// TwinCAT 3 PLC project Green_Crane
// ProgramVersion: 3.1.4023.0
// libraries:
//   Tc2_Standard, * (Beckhoff Automation GmbH)
//   Tc2_System, * (Beckhoff Automation GmbH)
//   Tc3_Module, * (Beckhoff Automation GmbH)
// project tree:
//   DUTs/ E_Mode.TcDUT, ST_ActiveDamping.TcDUT
//   / GlobalTextList.TcGTLO, PlcTask.TcTTO, Visualization Manager.TcVMO (not stored)
//   GVLs/ G_Input.TcGVL, G_Output.TcGVL, G_Parameter.TcGVL
//   POUs/FBs/ FB_AutomaticControl.TcPOU, FB_Clock.TcPOU, FB_ManualControl.TcPOU, FB_SetMode.TcPOU
//   POUs/Imported FBs/ FB_CraneSimulator.TcPOU, FB_MotionReferenceGenerat.TcPOU, FB_ActiveDamping.TcPOU, FB_ClosedLoopControl.TcPOU, FB_OpenLoopControl.TcPOU, FB_ResetIntegralController.TcPOU
//   POUs/Programs/ MAIN.TcPOU (not stored), P_CraneControl.TcPOU
//   VISUs/ HMI.TcVIS
// real-time tasks:
//   TASK PlcTask: cycle T#10ms, priority 20, ADS port 350

CONFIGURATION Green_Crane
    RESOURCE PLC ON TwinCAT3
        TASK PlcTask(INTERVAL := T#10ms, PRIORITY := 20);
        PROGRAM MAIN WITH PlcTask : MAIN;
    END_RESOURCE
END_CONFIGURATION

// ---- DUTs/E_Mode.TcDUT
{attribute 'qualified_only'}
{attribute 'strict'}
TYPE E_Mode :
(
	Auto,
	Manual,
	Off
);
END_TYPE

// ---- DUTs/ST_ActiveDamping.TcDUT
TYPE ST_ActiveDamping :
STRUCT
	fFlowGainInverse : LREAL := 1.7153E03;	
	fHPF_Num1 : LREAL := 9.016E-12;
	fHPF_Num2 : LREAL := -9.016E-12;
	fHPF_Den1 : LREAL := 1.0;
	fHPF_Den2 : LREAL := -0.9905;
	fVDI_Num1 : LREAL := 25;
	fVDI_Num2 : LREAL := -48.83;
	fVDI_Num3 : LREAL := 23.85;
	fVDI_Den1 : LREAL := 1;
	fVDI_Den2 : LREAL := -1.721;
	fVDI_Den3 : LREAL := 0.7408;
END_STRUCT
END_TYPE

// ---- GVLs/G_Input.TcGVL
{attribute 'qualified_only'}
VAR_GLOBAL
	bPoweSwitch : BOOL;
	bOnOffSwitch : BOOL;
	bModeSwitch : BOOL;
	bStartSwitch : BOOL;
	bStopSwitch : BOOL;
	fJoyStickSignal : REAL;
END_VAR

// ---- GVLs/G_Output.TcGVL
{attribute 'qualified_only'}
VAR_GLOBAL
	sModeDisplay : STRING;
	bGreenLed : BOOL;
	bRedLed : BOOL;
	fOpenLoopControlOutput : LREAL;
	
END_VAR

// ---- GVLs/G_Parameter.TcGVL
{attribute 'qualified_only'}
VAR_GLOBAL
	fCycleTime : REAL := 0.01;
	fTime : REAL;
	eMode : E_Mode;
	fMaxVolumeFlow : REAL := 30.0;
	fCylinderSpeedRef : LREAL;
	
	
// MotionReference
	fStartPosition_m		: LREAL := 0.0;
	fStartVelocity_m		: LREAL	:= 0.0;
	fPositionSetpoint_ms	: LREAL := 0.25;
	fVelocitySetpoint_m		: LREAL := 0.025;
	fMaxPosition 			: LREAL := 0.45;
	fMinPosition 			: LREAL := 0.0;
	fMaxVelocity 			: LREAL := 0.05;
	fTimeBeforeStarting_s	: LREAL := 3.0;
	fRampTime_s				: LREAL := 1.0;
	fHoldPositionTime_s		: LREAL := 5.0;




// Automatic

	bEnableVelocityFeedForwardControl	: BOOL := TRUE;
	bEnableClosedLoopPositionControl	: BOOL := TRUE;
	bEnableIntegralController 			: BOOL := TRUE;
	bEnableActiveDamping 				: BOOL := TRUE;


// Closed Loop
	fMaxPositionError 					: LREAL := 1E-3;
	fProportionalGain 					: LREAL := 29.17;
	fIntegralGain 						: LREAL := 19.49;	
	
	
//Simulator

	bEnableSimulation					: BOOL := TRUE;
	
END_VAR

// ---- POUs/FBs/FB_AutomaticControl.TcPOU
FUNCTION_BLOCK FB_AutomaticControl
VAR_INPUT
	bEnable : BOOL;
	eMode : E_Mode;
	bStartSwitch : BOOL;
	bStopSwitch : BOOL;
END_VAR
VAR_OUTPUT
	fAutoOutput : LREAL;
END_VAR
VAR
	fbClock 						: FB_Clock;
	fbMotionReference 				: FB_MotionReferenceGenerat;
	fbVelocityFeedForwardControl 	: FB_OpenLoopControl;
	fbResetIntegralController		: FB_ResetIntegralController;
	fbClosedLoopControl		: FB_ClosedLoopControl;
	
	
	fStartPosition : LREAL;
	fStartVelocity : LREAL;
	fPositionSetpoint : LREAL;
	fVelocitySetpoint : LREAL;
	fTimeBeforeStarting : LREAL;
	fRampTime : LREAL;
	fHoldPositionTime : LREAL;

END_VAR

IF bEnable = FALSE THEN
	RETURN;
END_IF


fbClock(
	bStart := ((eMode = E_Mode.Auto) AND bStartSwitch = TRUE),
	bStop := bStopSwitch,
	fCycleTime := G_Parameter.fCycleTime,
);

fStartPosition := LIMIT(G_Parameter.fMinPosition, G_parameter.fStartPosition_m, G_Parameter.fMaxPosition);
fStartVelocity := LIMIT(0.0, G_parameter.fStartVelocity_m, G_parameter.fMaxVelocity );
fPositionSetpoint := LIMIT(G_Parameter.fMinPosition, G_Parameter.fPositionSetpoint_ms, G_Parameter.fMaxPosition);
fVelocitySetpoint := LIMIT(0.0, G_Parameter.fVelocitySetpoint_m, G_Parameter.fMaxVelocity);
fTimeBeforeStarting := LIMIT(0.0, G_Parameter.fTimeBeforeStarting_s, 10.0);
fRampTime := LIMIT(0.0, G_Parameter.fRampTime_s, 10.0);
fHoldPositionTime := LIMIT(0.0, G_Parameter.fHoldPositionTime_s, 60.0);

fbMotionReference(
	fStartposition_m := fStartPosition,
	fStartVelocity_m := fStartVelocity,
	fPositionSetpoint_ms := fPositionSetpoint,
	fVelocitySetpoint_m := fVelocitySetpoint,
	fTimeBeforeStarting_s := fTimeBeforeStarting,
	fRampTime_s := fRampTime,
	fHoldPositionTime_s := fHoldPositionTime,
	fClock_s := fbClock.fTimeInSeconds
);
	
	
fbVelocityFeedForwardControl(
	bEnable := G_Parameter.bEnableVelocityFeedForwardControl,
	fVelocityReference_ms := fbMotionReference.fVelocityReference_ms,
	fMaxValveFlow_lmin := G_Parameter.fMaxVolumeFlow
);
		
fbResetIntegralController(
	fVelocityReference_ms := fbMotionReference.fVelocityReference_ms,
	fPositionError_m := fbClosedLoopControl.fPositionError,
	fMaxPositionError_m := G_Parameter.fMaxPosition
);
	
	

fbClosedLoopControl(
	bEnable := G_Parameter.bEnableClosedLoopPositionControl,
	bActivateIntegralController := G_Parameter.bEnableIntegralController,
	bIntegralControllReset := fbResetIntegralController.bReset,
	fPositionFeedBack := 0.0,
	fProportionalGain := G_Parameter.fProportionalGain,
	fPositionReference := fbMotionReference.fPositionReference_m,
);
	
	IF (eMode = E_Mode.Auto AND G_input.bStartSwitch = TRUE) THEN
	fAutoOutput := LIMIT(-1.0, (fbVelocityFeedForwardControl.fVelocityFeedForward + fbClosedLoopControl.fClosedLoopPosition), 1.0);
ELSE
	fAutoOutput:= 0.0;
END_IF

END_FUNCTION_BLOCK

// ---- POUs/FBs/FB_Clock.TcPOU
FUNCTION_BLOCK FB_Clock
VAR_INPUT
	bStart : BOOL;
	bStop : BOOL;
	fCycleTime : REAL;
END_VAR
VAR_OUTPUT
	fTimeInSeconds : REAL;
END_VAR
VAR
END_VAR



IF bStart = TRUE AND bStop = FALSE THEN
	fTimeInSeconds := fTimeInSeconds + fCycleTime;
ELSE
	fTimeInSeconds := 0.0;
END_IF

END_FUNCTION_BLOCK

// ---- POUs/Imported FBs/FB_MotionReferenceGenerat.TcPOU
FUNCTION_BLOCK FB_MotionReferenceGenerat
VAR_INPUT
	fStartPosition_m: LREAL;
	fStartVelocity_m: LREAL;
	fPositionSetpoint_ms: LREAL;
	fVelocitySetpoint_m: LREAL;
	fTimeBeforeStarting_s: LREAL;
	fRampTime_s: LREAL;
	fHoldPositionTime_s: LREAL;
	fClock_s: LREAL;
END_VAR
VAR_OUTPUT
	fPositionReference_m: LREAL;
	fVelocityReference_ms: LREAL;
	fTotalMotionTime_s: LREAL;
	fErrorSignal: LREAL;
END_VAR
VAR
	Error: DINT;
	slopeExt: LREAL;
	slopeRetr: LREAL;
	tHold: LREAL;
	x1: LREAL;
	x4: LREAL;
	x1_tmp: LREAL;
	x1_tmp_tmp: LREAL;
	x4_tmp: LREAL;
	x4_tmp_tmp: LREAL;
	x4_tmp_tmp_0: LREAL;
	x1_tmp_0: LREAL;
END_VAR


(* Outputs for Atomic SubSystem: '<Root>/FB_MotionReferenceGenerator_nolimit' *)
(* MATLAB Function: '<S1>/WaveSignal' *)
(* MATLAB Function 'FB_MotionReferenceGenerator_nolimit/WaveSignal': '<S2>:1' *)
(* '<S2>:1:2' x_SP = x_ref - x0; *)
(* '<S2>:1:3' vs=v_ref; *)
(* '<S2>:1:4' slopeExt=v0-vs; *)
slopeExt := fStartVelocity_m - fVelocitySetpoint_m;
(* '<S2>:1:5' slopeRetr=-vs-v0; *)
slopeRetr := ( -fVelocitySetpoint_m) - fStartVelocity_m;
(* '<S2>:1:7' as = vs/tRamp; *)
(* '<S2>:1:8' s_acc=(vs^2-v0^2)/as; *)
(* '<S2>:1:10' tHold=(x_SP-s_acc)/vs; *)
tHold := ((fPositionSetpoint_ms - fStartPosition_m) - (((fVelocitySetpoint_m * fVelocitySetpoint_m) - (fStartVelocity_m * fStartVelocity_m)) / (fVelocitySetpoint_m / fRampTime_s))) / fVelocitySetpoint_m;
(* '<S2>:1:12' if tHold < 0 *)

IF tHold < 0.0 THEN 
    (* '<S2>:1:13' Error = 1; *)
    Error := 1;
ELSE 
    (* '<S2>:1:14' else *)
    (* '<S2>:1:15' Error = 0; *)
    Error := 0;
END_IF;

(* '<S2>:1:18' t1=tRamp; *)
(* '<S2>:1:19' t2=tHold; *)
(* '<S2>:1:20' t3=tRamp; *)
(* '<S2>:1:21' t4=tWait; *)
(* '<S2>:1:22' t5=t1; *)
(* '<S2>:1:23' t6=t2; *)
(* '<S2>:1:24' t7=t3; *)
(* '<S2>:1:26' x = x0; *)
(* '<S2>:1:27' x1 = x0 + v0*((t0+t1)-t0)-(slopeExt/t1)*((t0+t1)-t0)^2/2; *)
x1_tmp_tmp := fTimeBeforeStarting_s + fRampTime_s;
x1_tmp := x1_tmp_tmp - fTimeBeforeStarting_s;
x1_tmp_0 := slopeExt / fRampTime_s;
x1 := ((x1_tmp * fStartVelocity_m) + fStartPosition_m) - ((x1_tmp_0 * (x1_tmp * x1_tmp)) / 2.0);
(* '<S2>:1:28' x2 = x1 + vs*((t0+t1+t2)-(t0+t1)); *)
(* '<S2>:1:29' x4 = x_ref - v0*((t0+t1+t2+t3+t4+t5)-(t0+t1+t2+t3+t4))+(slopeRetr/t5)*((t0+t1+t2+t3+t4+t5)-(t0+t1+t2+t3+t4))^2/2; *)
x4_tmp_tmp := x1_tmp_tmp + tHold;
x4_tmp_tmp_0 := x4_tmp_tmp + fRampTime_s;
x4_tmp := x4_tmp_tmp_0 + fHoldPositionTime_s;
x1_tmp := x4_tmp + fRampTime_s;
x4 := x1_tmp - x4_tmp;
x4 := (fPositionSetpoint_ms - (x4 * fStartVelocity_m)) + (((slopeRetr / fRampTime_s) * (x4 * x4)) / 2.0);
(* '<S2>:1:30' x5 = x4-vs*((t0+t1+t2+t3+t4+t5+t6)-(t0+t1+t2+t3+t4+t5)); *)
(* '<S2>:1:32' if Error == 1 *)

IF Error = 1 THEN 
    (* Outport: '<Root>/fPositionReference_m' *)
    (* '<S2>:1:33' x = x0; *)
    fPositionReference_m := fStartPosition_m;
    (* Outport: '<Root>/fVelocityReference_ms' *)
    (* '<S2>:1:34' v = v0; *)
    fVelocityReference_ms := fStartVelocity_m;
ELSIF (fClock_s >= 0.0) AND (fClock_s < fTimeBeforeStarting_s) THEN 
    (* Outport: '<Root>/fPositionReference_m' *)
    (* '<S2>:1:35' elseif t>=0 && t<t0 *)
    (* '<S2>:1:36' x = x0; *)
    fPositionReference_m := fStartPosition_m;
    (* Outport: '<Root>/fVelocityReference_ms' *)
    (* '<S2>:1:37' v = v0; *)
    fVelocityReference_ms := fStartVelocity_m;
ELSIF (fClock_s >= fTimeBeforeStarting_s) AND (fClock_s < x1_tmp_tmp) THEN 
    (* '<S2>:1:38' elseif t>=t0 && t<(t0+t1) *)
    (* '<S2>:1:39' x = x0 + v0*(t-t0)-(slopeExt/t1)*(t-t0)^2/2; *)
    slopeRetr := fClock_s - fTimeBeforeStarting_s;
    (* Outport: '<Root>/fPositionReference_m' *)
    fPositionReference_m := ((slopeRetr * fStartVelocity_m) + fStartPosition_m) - ((x1_tmp_0 * (slopeRetr * slopeRetr)) / 2.0);
    (* Outport: '<Root>/fVelocityReference_ms' *)
    (* '<S2>:1:40' v = v0-(slopeExt/t1)*(t-t0); *)
    fVelocityReference_ms := fStartVelocity_m - (x1_tmp_0 * slopeRetr);
ELSIF (fClock_s >= x1_tmp_tmp) AND (fClock_s < x4_tmp_tmp) THEN 
    (* Outport: '<Root>/fPositionReference_m' *)
    (* '<S2>:1:41' elseif t>=(t0+t1) && t<(t0+t1+t2) *)
    (* '<S2>:1:42' x = x1 + vs*(t-(t0+t1)); *)
    fPositionReference_m := ((fClock_s - x1_tmp_tmp) * fVelocitySetpoint_m) + x1;
    (* Outport: '<Root>/fVelocityReference_ms' *)
    (* '<S2>:1:43' v = vs; *)
    fVelocityReference_ms := fVelocitySetpoint_m;
ELSIF (fClock_s >= x4_tmp_tmp) AND (fClock_s < x4_tmp_tmp_0) THEN 
    (* '<S2>:1:44' elseif t>=(t0+t1+t2) && t<(t0+t1+t2+t3) *)
    (* '<S2>:1:45' x = x2+vs*(t-(t0+t1+t2))+(slopeExt/t3)*(t-(t0+t1+t2))^2/2; *)
    slopeRetr := fClock_s - x4_tmp_tmp;
    (* Outport: '<Root>/fPositionReference_m' *)
    fPositionReference_m := ((((x4_tmp_tmp - x1_tmp_tmp) * fVelocitySetpoint_m) + x1) + (slopeRetr * fVelocitySetpoint_m)) + ((x1_tmp_0 * (slopeRetr * slopeRetr)) / 2.0);
    (* Outport: '<Root>/fVelocityReference_ms' *)
    (* '<S2>:1:46' v = vs+(slopeExt/t3)*(t-(t0+t1+t2)); *)
    fVelocityReference_ms := (slopeRetr * (slopeExt / fRampTime_s)) + fVelocitySetpoint_m;
ELSIF (fClock_s >= x4_tmp_tmp_0) AND (fClock_s < x4_tmp) THEN 
    (* Outport: '<Root>/fPositionReference_m' *)
    (* '<S2>:1:47' elseif t>=(t0+t1+t2+t3) && t<(t0+t1+t2+t3+t4) *)
    (* '<S2>:1:48' x = x_ref; *)
    fPositionReference_m := fPositionSetpoint_ms;
    (* Outport: '<Root>/fVelocityReference_ms' *)
    (* '<S2>:1:49' v = v0; *)
    fVelocityReference_ms := fStartVelocity_m;
ELSIF (fClock_s >= x4_tmp) AND (fClock_s < x1_tmp) THEN 
    (* '<S2>:1:50' elseif t>=(t0+t1+t2+t3+t4) && t<(t0+t1+t2+t3+t4+t5) *)
    (* '<S2>:1:51' x = x_ref - v0*(t-(t0+t1+t2+t3+t4))+(slopeRetr/t5)*(t-(t0+t1+t2+t3+t4))^2/2; *)
    slopeExt := fClock_s - x4_tmp;
    slopeRetr := slopeRetr / fRampTime_s;
    (* Outport: '<Root>/fPositionReference_m' *)
    fPositionReference_m := (fPositionSetpoint_ms - (slopeExt * fStartVelocity_m)) + ((slopeRetr * (slopeExt * slopeExt)) / 2.0);
    (* Outport: '<Root>/fVelocityReference_ms' *)
    (* '<S2>:1:52' v = v0+(slopeRetr/t5)*(t-(t0+t1+t2+t3+t4)); *)
    fVelocityReference_ms := (slopeExt * slopeRetr) + fStartVelocity_m;
ELSE 
    x1_tmp_0 := x1_tmp + tHold;

    IF (fClock_s >= x1_tmp) AND (fClock_s < x1_tmp_0) THEN 
        (* Outport: '<Root>/fPositionReference_m' *)
        (* '<S2>:1:53' elseif t>=(t0+t1+t2+t3+t4+t5) && t<(t0+t1+t2+t3+t4+t5+t6) *)
        (* '<S2>:1:54' x = x4-vs*(t-(t0+t1+t2+t3+t4+t5)); *)
        fPositionReference_m := x4 - ((fClock_s - x1_tmp) * fVelocitySetpoint_m);
        (* Outport: '<Root>/fVelocityReference_ms' *)
        (* '<S2>:1:55' v = -vs; *)
        fVelocityReference_ms :=  -fVelocitySetpoint_m;
    ELSIF (fClock_s >= x1_tmp_0) AND (fClock_s < (((((((fTimeBeforeStarting_s + fRampTime_s) + tHold) + fRampTime_s) + fHoldPositionTime_s) + fRampTime_s) + tHold) + fRampTime_s)) THEN 
        (* '<S2>:1:56' elseif t>=(t0+t1+t2+t3+t4+t5+t6) && t<(t0+t1+t2+t3+t4+t5+t6+t7) *)
        (* '<S2>:1:57' x = x5-vs*(t-(t0+t1+t2+t3+t4+t5+t6))-(slopeRetr/t3)*(t-(t0+t1+t2+t3+t4+t5+t6))^2/2; *)
        slopeExt := fClock_s - x1_tmp_0;
        slopeRetr := slopeRetr / fRampTime_s;
        (* Outport: '<Root>/fPositionReference_m' *)
        fPositionReference_m := ((x4 - ((x1_tmp_0 - x1_tmp) * fVelocitySetpoint_m)) - (slopeExt * fVelocitySetpoint_m)) - ((slopeRetr * (slopeExt * slopeExt)) / 2.0);
        (* Outport: '<Root>/fVelocityReference_ms' *)
        (* '<S2>:1:58' v = -vs-(slopeRetr/t3)*(t-(t0+t1+t2+t3+t4+t5+t6)); *)
        fVelocityReference_ms := ( -fVelocitySetpoint_m) - (slopeExt * slopeRetr);
    ELSE 
        (* Outport: '<Root>/fPositionReference_m' *)
        (* '<S2>:1:59' else *)
        (* '<S2>:1:60' x = x0; *)
        fPositionReference_m := fStartPosition_m;
        (* Outport: '<Root>/fVelocityReference_ms' *)
        (* '<S2>:1:61' v = v0; *)
        fVelocityReference_ms := fStartVelocity_m;
    END_IF;

END_IF;

(* Outport: '<Root>/fTotalMotionTime_s' incorporates:
 *  MATLAB Function: '<S1>/WaveSignal' *)
(* '<S2>:1:64' T = t0+t1+t2+t3+t4+t5+t6+t7; *)
fTotalMotionTime_s := ((((((fTimeBeforeStarting_s + fRampTime_s) + tHold) + fRampTime_s) + fHoldPositionTime_s) + fRampTime_s) + tHold) + fRampTime_s;
(* Outport: '<Root>/fErrorSignal' incorporates:
 *  MATLAB Function: '<S1>/WaveSignal' *)
fErrorSignal := DINT_TO_LREAL(Error);
(* End of Outputs for SubSystem: '<Root>/FB_MotionReferenceGenerator_nolimit' *)

END_FUNCTION_BLOCK

// ---- POUs/Imported FBs/FB_OpenLoopControl.TcPOU
FUNCTION_BLOCK FB_OpenLoopControl
VAR_INPUT
	bEnable: BOOL;
	fVelocityReference_ms: LREAL;
	fMaxValveFlow_lmin: LREAL;
END_VAR
VAR_OUTPUT
	fVelocityFeedForward: LREAL;
END_VAR
VAR
END_VAR


(* Outputs for Atomic SubSystem: '<Root>/FB_OpenLoopControl' *)
(* Switch: '<S1>/Switch2' incorporates:
 *  Constant: '<S1>/Annnulus_Area'
 *  Constant: '<S1>/Bore_Area'
 *  Product: '<S1>/Product1'
 *  Product: '<S1>/Product3' *)

IF fVelocityReference_ms >= 0.0 THEN 
    fVelocityFeedForward := 0.0033183 * fVelocityReference_ms;
ELSE 
    fVelocityFeedForward := fVelocityReference_ms * 0.0023562;
END_IF;

(* End of Switch: '<S1>/Switch2' *)


(* Switch: '<S1>/Switch1' incorporates:
 *  Constant: '<S1>/Constant'
 *  Gain: '<S1>/Gain1'
 *  Product: '<S1>/Divide2' *)

IF bEnable THEN 
    fVelocityFeedForward := (60000.0 * fVelocityFeedForward) / fMaxValveFlow_lmin;
ELSE 
    fVelocityFeedForward := 0.0;
END_IF;

(* End of Switch: '<S1>/Switch1' *)


(* Saturate: '<S1>/Saturation1' *)

IF fVelocityFeedForward > 1.0 THEN 
    (* Outport: '<Root>/fVelocityFeedForward' *)
    fVelocityFeedForward := 1.0;
ELSIF fVelocityFeedForward < -1.0 THEN 
    (* Outport: '<Root>/fVelocityFeedForward' *)
    fVelocityFeedForward := -1.0;
END_IF;

(* End of Saturate: '<S1>/Saturation1' *)
(* End of Outputs for SubSystem: '<Root>/FB_OpenLoopControl' *)

END_FUNCTION_BLOCK

// ---- POUs/Imported FBs/FB_ResetIntegralController.TcPOU
FUNCTION_BLOCK FB_ResetIntegralController
VAR_INPUT
	fVelocityReference_ms: LREAL;
	fMaxPositionError_m: LREAL;
	fPositionError_m: LREAL;
END_VAR
VAR_OUTPUT
	bReset: BOOL;
END_VAR
VAR
	rtb_Reset: DINT;
END_VAR


(* Outputs for Atomic SubSystem: '<Root>/FB_ResetIntegralController' *)
(* MATLAB Function: '<S1>/ResetIntegralController' *)
(* MATLAB Function 'FB_ResetIntegralController/ResetIntegralController': '<S2>:1' *)
(* '<S2>:1:3' if abs(vRef) > 0 || abs(exCyl) > exCylMax *)

IF ABS(fVelocityReference_ms) > 0.0 THEN 
    (* '<S2>:1:4' Reset = 0; *)
    rtb_Reset := 0;
ELSIF ABS(fPositionError_m) > fMaxPositionError_m THEN 
    (* '<S2>:1:4' Reset = 0; *)
    rtb_Reset := 0;
ELSE 
    (* '<S2>:1:5' else *)
    (* '<S2>:1:6' Reset = 1; *)
    rtb_Reset := 1;
END_IF;

(* End of MATLAB Function: '<S1>/ResetIntegralController' *)


(* Outport: '<Root>/bReset' incorporates:
 *  DataTypeConversion: '<S1>/Data Type Conversion' *)
bReset := rtb_Reset <> 0;
(* End of Outputs for SubSystem: '<Root>/FB_ResetIntegralController' *)

END_FUNCTION_BLOCK

// ---- POUs/Imported FBs/FB_ClosedLoopControl.TcPOU
FUNCTION_BLOCK FB_ClosedLoopControl
VAR_INPUT

	bEnable: BOOL;
	bActivateIntegralController: BOOL;
	fProportionalGain: LREAL;
	fIntegralGain: LREAL;
	fPositionReference: LREAL;
	fPositionFeedback: LREAL;
	bIntegralControllReset: BOOL;
END_VAR
VAR_OUTPUT
	fClosedLoopPosition: LREAL;
	fPositionError: LREAL;
END_VAR
VAR
	rtb_u_FB: LREAL;
	rtb_Saturation1: LREAL;
	c_DiscreteTimeIntegrator_DS: LREAL;
END_VAR


        fPositionError := fPositionReference - fPositionFeedback;
        (* DiscreteIntegrator: '<S1>/Discrete-Time Integrator' *)

        IF bIntegralControllReset THEN 
            c_DiscreteTimeIntegrator_DS := 0.0;
        END_IF;


        IF c_DiscreteTimeIntegrator_DS >= 1.0 THEN 
            c_DiscreteTimeIntegrator_DS := 1.0;
        ELSIF c_DiscreteTimeIntegrator_DS <= -1.0 THEN 
            c_DiscreteTimeIntegrator_DS := -1.0;
        END_IF;

        (* Switch: '<S1>/Switch' incorporates:
         *  Constant: '<S1>/Constant'
         *  DiscreteIntegrator: '<S1>/Discrete-Time Integrator' *)

        IF bActivateIntegralController THEN 
            rtb_u_FB := c_DiscreteTimeIntegrator_DS;
        ELSE 
            rtb_u_FB := 0.0;
        END_IF;

        (* End of Switch: '<S1>/Switch' *)
        

        (* Sum: '<S1>/Sum5' incorporates:
         *  Product: '<S1>/Product' *)
        rtb_u_FB := (fProportionalGain * fPositionError) + rtb_u_FB;
        (* Saturate: '<S1>/Saturation1' *)

        IF rtb_u_FB > 1.0 THEN 
            rtb_Saturation1 := 1.0;
        ELSIF rtb_u_FB >= -1.0 THEN 
            rtb_Saturation1 := rtb_u_FB;
        ELSE 
            rtb_Saturation1 := -1.0;
        END_IF;

        (* End of Saturate: '<S1>/Saturation1' *)
        

        (* Switch: '<S1>/Switch1' *)

        IF bEnable THEN 
            (* Outport: '<Root>/fClosedLoopPosition' *)
            fClosedLoopPosition := rtb_Saturation1;
        ELSE 
            (* Outport: '<Root>/fClosedLoopPosition' incorporates:
             *  Constant: '<S1>/Constant1' *)
            fClosedLoopPosition := 0.0;
        END_IF;

        (* End of Switch: '<S1>/Switch1' *)
        

        (* Update for DiscreteIntegrator: '<S1>/Discrete-Time Integrator' incorporates:
         *  Product: '<S1>/Divide'
         *  Product: '<S1>/Product2'
         *  Sum: '<S1>/Sum2'
         *  Sum: '<S1>/Sum3' *)
        c_DiscreteTimeIntegrator_DS := (((((rtb_Saturation1 - rtb_u_FB) / fProportionalGain) + fPositionError) * fIntegralGain) * 0.01) + c_DiscreteTimeIntegrator_DS;

        IF c_DiscreteTimeIntegrator_DS >= 1.0 THEN 
            c_DiscreteTimeIntegrator_DS := 1.0;
        ELSIF c_DiscreteTimeIntegrator_DS <= -1.0 THEN 
            c_DiscreteTimeIntegrator_DS := -1.0;
        END_IF;

        (* End of Update for DiscreteIntegrator: '<S1>/Discrete-Time Integrator' *)
        (* End of Outputs for SubSystem: '<Root>/FB_ClosedLoopControl' *)

END_FUNCTION_BLOCK

// ---- POUs/FBs/FB_ManualControl.TcPOU
FUNCTION_BLOCK FB_ManualControl
VAR_INPUT
	bEnable : BOOL;
	eMode : E_Mode;
	fJoyStickInput : REAL;
END_VAR
VAR_OUTPUT
	fManualControlOutput : LREAL;
END_VAR
VAR
	fbOpenLoopControl : FB_OpenLoopControl;

;END_VAR


IF bEnable = FALSE THEN
	RETURN;
END_IF

G_Parameter.fCylinderSpeedRef := G_Parameter.fMaxVelocity * G_Input.fJoyStickSignal;

fbOpenLoopControl
(
	bEnable := (G_Parameter.eMode = E_Mode.Manual),
	fVelocityReference_ms := G_Parameter.fCylinderSpeedRef,
	fMaxValveFlow_lmin := G_Parameter.fMaxVolumeFlow,
	fVelocityFeedForward => fManualControlOutput	
);

END_FUNCTION_BLOCK

// ---- POUs/FBs/FB_SetMode.TcPOU
FUNCTION_BLOCK FB_SetMode
VAR_INPUT
	bPower : BOOL;
	bOn : BOOL;
	bMode : BOOL;
	bStart : BOOL;
	bStop : BOOL;
END_VAR
VAR_OUTPUT
	eMode : E_Mode;
	sMode : STRING;
	bGreenLight : BOOL;
	bRedLight : BOOL;
END_VAR
VAR
END_VAR



IF bPower = TRUE THEN	
	IF bON = FALSE OR bStart = FALSE OR bStop = TRUE THEN
		eMode		:=	E_Mode.Off;
		bGreenLight	:=	FALSE;
		bRedLight 	:=	TRUE;
	
	ELSIF bON = TRUE AND bStart = TRUE AND bSTOP = FALSE THEN
		IF bMode = FALSE THEN
		eMode := E_Mode.Manual;
		ELSE
		eMode := E_Mode.Auto;
		END_IF
		
	bGreenLight := TRUE;
	bRedLight := FALSE;
		
	END_IF
ELSE
		eMode := E_Mode.Off;
		bGreenLight := FALSE; // No power = No lights
		bRedLight := FALSE;	  // NO power = No lights
END_IF




// String to HMI displaying current mode
IF eMode = E_Mode.Auto THEN
	sMode := 'AUTO';
ELSIF eMode = E_Mode.Manual THEN
	sMode := 'Manual';

ELSE
	sMode := 'OFF';
END_IF

END_FUNCTION_BLOCK

// ---- POUs/Imported FBs/FB_CraneSimulator.TcPOU
FUNCTION_BLOCK FB_CraneSimulator
VAR_INPUT
	ssMethodType: SINT;
	uDCV: LREAL;
END_VAR
VAR_OUTPUT
	xm: LREAL;
	ppbar: LREAL;
	prbar: LREAL;
END_VAR
VAR
	pLS: LREAL;
	QDCV_out: LREAL;
	rtb_xDot: LREAL;
	rtb_xDotDot: LREAL;
	temp1: LREAL;
	temp2: LREAL;
	temp3: LREAL;
	temp4: LREAL;
	c_DiscreteTimeIntegrator2_D: LREAL;
	c_DiscreteTimeIntegrator3_D: LREAL;
	c_DiscreteTimeIntegrator_DS: LREAL;
	c_DiscreteTimeIntegrator4_D: LREAL;
END_VAR



CASE ssMethodType OF
    0: 
        (* SystemInitialize for Atomic SubSystem: '<Root>/FB_CraneSimulator' *)
        (* InitializeConditions for DiscreteIntegrator: '<S1>/Discrete-Time Integrator' *)
        c_DiscreteTimeIntegrator_DS := 4.377E+6;
        (* InitializeConditions for DiscreteIntegrator: '<S1>/Discrete-Time Integrator2' *)
        c_DiscreteTimeIntegrator2_D := 0.0;
        (* InitializeConditions for DiscreteIntegrator: '<S1>/Discrete-Time Integrator3' *)
        c_DiscreteTimeIntegrator3_D := 0.0;
        (* InitializeConditions for DiscreteIntegrator: '<S1>/Discrete-Time Integrator4' *)
        c_DiscreteTimeIntegrator4_D := 468300.0;
        (* End of SystemInitialize for SubSystem: '<Root>/FB_CraneSimulator' *)
    1: 
        (* Outputs for Atomic SubSystem: '<Root>/FB_CraneSimulator' *)
        (* DiscreteIntegrator: '<S1>/Discrete-Time Integrator2' *)
        rtb_xDot := c_DiscreteTimeIntegrator2_D;
        (* Outport: '<Root>/x [m]' incorporates:
         *  DiscreteIntegrator: '<S1>/Discrete-Time Integrator3' *)
        xm := c_DiscreteTimeIntegrator3_D;
        (* Outport: '<Root>/pp [bar]' incorporates:
         *  DiscreteIntegrator: '<S1>/Discrete-Time Integrator'
         *  Gain: '<S1>/Gain' *)
        ppbar := 1.0E-5 * c_DiscreteTimeIntegrator_DS;
        (* Outport: '<Root>/pr [bar]' incorporates:
         *  DiscreteIntegrator: '<S1>/Discrete-Time Integrator4'
         *  Gain: '<S1>/Gain1' *)
        prbar := 1.0E-5 * c_DiscreteTimeIntegrator4_D;
        (* MATLAB Function: '<S1>/MATLAB Function' incorporates:
         *  DiscreteIntegrator: '<S1>/Discrete-Time Integrator'
         *  DiscreteIntegrator: '<S1>/Discrete-Time Integrator2'
         *  DiscreteIntegrator: '<S1>/Discrete-Time Integrator3'
         *  DiscreteIntegrator: '<S1>/Discrete-Time Integrator4' *)
        (* Parameters *)
        (* MATLAB Function 'FB_CraneSimulator/MATLAB Function': '<S2>:1' *)
        (* '<S2>:1:3' Fexternal = 1.3365e+04; *)
        (* [N] *)
        (* '<S2>:1:4' mEffective = 1.3365e+04; *)
        (* [kg] *)
        (* '<S2>:1:5' kFric = 4000; *)
        (* [N/(ms)] *)
        (* '<S2>:1:6' Apiston = 0.0033; *)
        (* [m^2] *)
        (* '<S2>:1:7' Aannulus = 0.0023; *)
        (* [m^2] *)
        (* '<S2>:1:8' beta = 1.0e9; *)
        (* [Pa] *)
        (* '<S2>:1:9' pSupply = 180e5; *)
        (* [Pa] *)
        (* '<S2>:1:10' pReturn = 1.1e5; *)
        (* [Pa] *)
        (* '<S2>:1:11' MaxStroke = 0.5; *)
        (* [m] *)
        (* '<S2>:1:12' VCyl_A = 1.0e-03; *)
        (* '<S2>:1:13' VCyl_B = 1.25e-03; *)
        (* '<S2>:1:14' p_nom_DCV = 7e5; *)
        (* '<S2>:1:15' Q1_ref_DCV = 20/6e4; *)
        (* '<S2>:1:16' kv1_DCV = Q1_ref_DCV/sqrt(p_nom_DCV); *)
        (* '<S2>:1:17' p0 = 7e5; *)
        (* compensator crack pressure *)
        (* Directional Control Valve - Lifting Cylinder  *)
        (* LS Pressure *)
        (* '<S2>:1:20' if uDCV > 0 *)

        IF uDCV > 0.0 THEN 
            (* '<S2>:1:21' pLS = pPiston; *)
            pLS := c_DiscreteTimeIntegrator_DS;
        ELSIF uDCV < 0.0 THEN 
            (* '<S2>:1:22' elseif uDCV < 0 *)
            (* '<S2>:1:23' pLS = pRod; *)
            pLS := c_DiscreteTimeIntegrator4_D;
        ELSE 
            (* '<S2>:1:24' else *)
            (* '<S2>:1:25' pLS = 0; *)
            pLS := 0.0;
        END_IF;

        (* '<S2>:1:28' if pLS<0 *)

        IF pLS < 0.0 THEN 
            (* '<S2>:1:29' pLS = 0; *)
            pLS := 0.0;
        END_IF;

        (* Pressure Compensator *)
        (* '<S2>:1:33' pPC = 0; *)
        (* '<S2>:1:35' if p0 <= (pSupply - pLS) *)

        IF 700000.0 <= (1.8E+7 - pLS) THEN 
            (* '<S2>:1:36' pPC = pLS+p0; *)
            pLS := pLS + 700000.0;
        ELSE 
            (* '<S2>:1:37' elseif 0 < (pSupply - pLS) < p0 *)
            (* '<S2>:1:38' pPC = pSupply-pLS; *)
            pLS := 1.8E+7 - pLS;
        END_IF;

        (* '<S2>:1:43' if pPC<0 *)

        IF pLS < 0.0 THEN 
            (* '<S2>:1:44' pPC = 0; *)
            pLS := 0.0;
        END_IF;

        (* Orifice Equations *)
        (* '<S2>:1:47' if uDCV > 0 *)

        IF uDCV > 0.0 THEN 
            (* '<S2>:1:48' QDCV_in =  kv1_DCV*uDCV*sign(pPC-pPiston)*sqrt(abs(pPC-pPiston)); *)
            pLS := pLS - c_DiscreteTimeIntegrator_DS;

            IF pLS < 0.0 THEN 
                rtb_xDotDot := -1.0;
            ELSIF pLS > 0.0 THEN 
                rtb_xDotDot := 1.0;
            ELSE 
                rtb_xDotDot := pLS;
            END_IF;

            temp3 := ABS(pLS);
            pLS := ((3.9840953644479785E-7 * uDCV) * rtb_xDotDot) * SQRT(temp3);
            (* '<S2>:1:49' QDCV_out = kv1_DCV*uDCV*sign(pRod-pReturn)*sqrt(abs(pRod-pReturn)); *)

            IF (c_DiscreteTimeIntegrator4_D - 110000.0) < 0.0 THEN 
                rtb_xDotDot := -1.0;
            ELSIF (c_DiscreteTimeIntegrator4_D - 110000.0) > 0.0 THEN 
                rtb_xDotDot := 1.0;
            ELSE 
                rtb_xDotDot := c_DiscreteTimeIntegrator4_D - 110000.0;
            END_IF;

            temp4 := ABS(c_DiscreteTimeIntegrator4_D - 110000.0);
            QDCV_out := ((3.9840953644479785E-7 * uDCV) * rtb_xDotDot) * SQRT(temp4);
        ELSIF uDCV < 0.0 THEN 
            (* '<S2>:1:50' elseif uDCV < 0 *)
            (* '<S2>:1:51' QDCV_out =  kv1_DCV*uDCV*sign(pPC-pRod)*sqrt(abs(pPC-pRod)); *)
            pLS := pLS - c_DiscreteTimeIntegrator4_D;

            IF pLS < 0.0 THEN 
                rtb_xDotDot := -1.0;
            ELSIF pLS > 0.0 THEN 
                rtb_xDotDot := 1.0;
            ELSE 
                rtb_xDotDot := pLS;
            END_IF;

            temp1 := ABS(pLS);
            QDCV_out := ((3.9840953644479785E-7 * uDCV) * rtb_xDotDot) * SQRT(temp1);
            (* '<S2>:1:52' QDCV_in =  kv1_DCV*uDCV*sign(pRod-pReturn)*sqrt(abs(pRod-pReturn)); *)

            IF (c_DiscreteTimeIntegrator4_D - 110000.0) < 0.0 THEN 
                rtb_xDotDot := -1.0;
            ELSIF (c_DiscreteTimeIntegrator4_D - 110000.0) > 0.0 THEN 
                rtb_xDotDot := 1.0;
            ELSE 
                rtb_xDotDot := c_DiscreteTimeIntegrator4_D - 110000.0;
            END_IF;

            temp2 := ABS(c_DiscreteTimeIntegrator4_D - 110000.0);
            pLS := ((3.9840953644479785E-7 * uDCV) * rtb_xDotDot) * SQRT(temp2);
        ELSE 
            (* '<S2>:1:53' else *)
            (* '<S2>:1:54' QDCV_in = 0; *)
            pLS := 0.0;
            (* '<S2>:1:55' QDCV_out = 0; *)
            QDCV_out := 0.0;
        END_IF;

        (* Pressure Gradients *)
        (* '<S2>:1:58' VA = VCyl_A + x*Apiston; *)
        (* '<S2>:1:59' VB =  VCyl_B + (MaxStroke - x)*Aannulus; *)
        (* '<S2>:1:60' VA_dot = Apiston*xDot; *)
        (* '<S2>:1:61' VB_dot = -Aannulus*xDot; *)
        (* '<S2>:1:62' pPistonDot = beta/VA*(QDCV_in - VA_dot); *)
        (* '<S2>:1:63' pRodDot = beta/VB*(-QDCV_out - VB_dot); *)
        QDCV_out := (1.0E+9 / (((0.5 - c_DiscreteTimeIntegrator3_D) * 0.0023) + 0.00125)) * (( -QDCV_out) - (-0.0023 * c_DiscreteTimeIntegrator2_D));
        (* Viscouse Friction *)
        (* '<S2>:1:66' Ffric = kFric*xDot; *)
        (* Hydraulic Force *)
        (* '<S2>:1:69' Fhyd = pPiston*Apiston - pRod*Aannulus; *)
        (* Newton Second Law of Motion *)
        (* '<S2>:1:72' xDotDot = (Fhyd - Ffric - Fexternal)/mEffective; *)
        rtb_xDotDot := ((((c_DiscreteTimeIntegrator_DS * 0.0033) - (c_DiscreteTimeIntegrator4_D * 0.0023)) - (4000.0 * c_DiscreteTimeIntegrator2_D)) - 13365.0) / 13365.0;
        (* Update for DiscreteIntegrator: '<S1>/Discrete-Time Integrator' incorporates:
         *  DiscreteIntegrator: '<S1>/Discrete-Time Integrator2'
         *  DiscreteIntegrator: '<S1>/Discrete-Time Integrator3'
         *  MATLAB Function: '<S1>/MATLAB Function' *)
        c_DiscreteTimeIntegrator_DS := (((1.0E+9 / ((c_DiscreteTimeIntegrator3_D * 0.0033) + 0.001)) * (pLS - (0.0033 * c_DiscreteTimeIntegrator2_D))) * 0.0001) + c_DiscreteTimeIntegrator_DS;

        IF c_DiscreteTimeIntegrator_DS >= 1.8E+7 THEN 
            c_DiscreteTimeIntegrator_DS := 1.8E+7;
        ELSIF c_DiscreteTimeIntegrator_DS <= 110000.0 THEN 
            c_DiscreteTimeIntegrator_DS := 110000.0;
        END_IF;

        (* End of Update for DiscreteIntegrator: '<S1>/Discrete-Time Integrator' *)
        

        (* Update for DiscreteIntegrator: '<S1>/Discrete-Time Integrator2' *)
        c_DiscreteTimeIntegrator2_D := (0.0001 * rtb_xDotDot) + c_DiscreteTimeIntegrator2_D;

        IF c_DiscreteTimeIntegrator2_D >= 0.12 THEN 
            c_DiscreteTimeIntegrator2_D := 0.12;
        ELSIF c_DiscreteTimeIntegrator2_D <= -0.12 THEN 
            c_DiscreteTimeIntegrator2_D := -0.12;
        END_IF;

        (* End of Update for DiscreteIntegrator: '<S1>/Discrete-Time Integrator2' *)
        

        (* Update for DiscreteIntegrator: '<S1>/Discrete-Time Integrator3' *)
        c_DiscreteTimeIntegrator3_D := (0.0001 * rtb_xDot) + c_DiscreteTimeIntegrator3_D;

        IF c_DiscreteTimeIntegrator3_D >= 0.5 THEN 
            c_DiscreteTimeIntegrator3_D := 0.5;
        ELSIF c_DiscreteTimeIntegrator3_D <= 0.0 THEN 
            c_DiscreteTimeIntegrator3_D := 0.0;
        END_IF;

        (* End of Update for DiscreteIntegrator: '<S1>/Discrete-Time Integrator3' *)
        

        (* Update for DiscreteIntegrator: '<S1>/Discrete-Time Integrator4' *)
        c_DiscreteTimeIntegrator4_D := (0.0001 * QDCV_out) + c_DiscreteTimeIntegrator4_D;

        IF c_DiscreteTimeIntegrator4_D >= 1.8E+7 THEN 
            c_DiscreteTimeIntegrator4_D := 1.8E+7;
        ELSIF c_DiscreteTimeIntegrator4_D <= 110000.0 THEN 
            c_DiscreteTimeIntegrator4_D := 110000.0;
        END_IF;

        (* End of Update for DiscreteIntegrator: '<S1>/Discrete-Time Integrator4' *)
        (* End of Outputs for SubSystem: '<Root>/FB_CraneSimulator' *)
END_CASE;

END_FUNCTION_BLOCK

// ---- POUs/Imported FBs/FB_ActiveDamping.TcPOU
FUNCTION_BLOCK FB_ActiveDamping
VAR_INPUT
	ssMethodType: SINT;
	bEnable: BOOL;
	fPressurePistonSide_Pa: LREAL;
	fPressureRodSide_Pa: LREAL;
	fkQfInv: LREAL;
	HPF_Num1: LREAL;
	HPF_Num2: LREAL;
	HPF_Den1: LREAL;
	HPF_Den2: LREAL;
	VDI_Num1: LREAL;
	VDI_Num2: LREAL;
	VDI_Num3: LREAL;
	VDI_Den1: LREAL;
	VDI_Den2: LREAL;
	VDI_Den3: LREAL;
END_VAR
VAR_OUTPUT
	fPressureFeedback: LREAL;
END_VAR
VAR
	rtb_Switch3: LREAL;
	HighPassFilter_tmp: LREAL;
	VectorConcatenate: ARRAY[0..1] OF LREAL;
	VectorConcatenate1: ARRAY[0..1] OF LREAL;
	VectorConcatenate2: ARRAY[0..2] OF LREAL;
	VectorConcatenate3: ARRAY[0..2] OF LREAL;
	HighPassFilter_states: LREAL;
	ValveDynamicsInverse_states: ARRAY[0..1] OF LREAL;
END_VAR



CASE ssMethodType OF
    0: 
        (* SystemInitialize for Atomic SubSystem: '<Root>/FB_ActiveDamping' *)
        (* InitializeConditions for DiscreteTransferFcn: '<S1>/HighPassFilter' *)
        HighPassFilter_states := 0.0;
        (* InitializeConditions for DiscreteTransferFcn: '<S1>/ValveDynamicsInverse' *)
        ValveDynamicsInverse_states[0] := 0.0;
        ValveDynamicsInverse_states[1] := 0.0;
        (* End of SystemInitialize for SubSystem: '<Root>/FB_ActiveDamping' *)
    1: 
        (* Outputs for Atomic SubSystem: '<Root>/FB_ActiveDamping' *)
        (* Switch: '<S1>/Switch3' incorporates:
         *  Constant: '<S1>/Constant1'
         *  Constant: '<S1>/Constant2' *)

        IF bEnable THEN 
            rtb_Switch3 := 0.0;
        ELSE 
            rtb_Switch3 := 1.0;
        END_IF;

        (* End of Switch: '<S1>/Switch3' *)
        

        (* SignalConversion: '<S1>/ConcatBufferAtVector ConcatenateIn1' incorporates:
         *  Concatenate: '<S1>/Vector Concatenate' *)
        VectorConcatenate[0] := HPF_Num1;
        (* SignalConversion: '<S1>/ConcatBufferAtVector ConcatenateIn2' incorporates:
         *  Concatenate: '<S1>/Vector Concatenate' *)
        VectorConcatenate[1] := HPF_Num2;
        (* SignalConversion: '<S1>/ConcatBufferAtVector Concatenate1In1' incorporates:
         *  Concatenate: '<S1>/Vector Concatenate1' *)
        VectorConcatenate1[0] := HPF_Den1;
        (* SignalConversion: '<S1>/ConcatBufferAtVector Concatenate1In2' incorporates:
         *  Concatenate: '<S1>/Vector Concatenate1' *)
        VectorConcatenate1[1] := HPF_Den2;
        (* SignalConversion: '<S1>/ConcatBufferAtVector Concatenate2In1' incorporates:
         *  Concatenate: '<S1>/Vector Concatenate2' *)
        VectorConcatenate2[0] := VDI_Num1;
        (* SignalConversion: '<S1>/ConcatBufferAtVector Concatenate2In2' incorporates:
         *  Concatenate: '<S1>/Vector Concatenate2' *)
        VectorConcatenate2[1] := VDI_Num2;
        (* SignalConversion: '<S1>/ConcatBufferAtVector Concatenate2In3' incorporates:
         *  Concatenate: '<S1>/Vector Concatenate2' *)
        VectorConcatenate2[2] := VDI_Num3;
        (* SignalConversion: '<S1>/ConcatBufferAtVector Concatenate3In1' incorporates:
         *  Concatenate: '<S1>/Vector Concatenate3' *)
        VectorConcatenate3[0] := VDI_Den1;
        (* SignalConversion: '<S1>/ConcatBufferAtVector Concatenate3In2' incorporates:
         *  Concatenate: '<S1>/Vector Concatenate3' *)
        VectorConcatenate3[1] := VDI_Den2;
        (* SignalConversion: '<S1>/ConcatBufferAtVector Concatenate3In3' incorporates:
         *  Concatenate: '<S1>/Vector Concatenate3' *)
        VectorConcatenate3[2] := VDI_Den3;
        (* DiscreteTransferFcn: '<S1>/HighPassFilter' incorporates:
         *  Gain: '<S1>/muC'
         *  Sum: '<S1>/Add' *)

        IF rtb_Switch3 <> 0.0 THEN 
            HighPassFilter_states := 0.0;
        END_IF;

        HighPassFilter_tmp := (fPressurePistonSide_Pa - (0.7101 * fPressureRodSide_Pa)) - (VectorConcatenate1[1] * HighPassFilter_states);
        (* Product: '<S1>/Product' incorporates:
         *  DiscreteTransferFcn: '<S1>/HighPassFilter' *)
        fPressureFeedback := ((VectorConcatenate[0] * HighPassFilter_tmp) + (VectorConcatenate[1] * HighPassFilter_states)) * fkQfInv;
        (* Saturate: '<S1>/Saturation1' *)

        IF fPressureFeedback > 1.0 THEN 
            fPressureFeedback := 1.0;
        ELSIF fPressureFeedback < -1.0 THEN 
            fPressureFeedback := -1.0;
        END_IF;

        (* End of Saturate: '<S1>/Saturation1' *)
        

        (* DiscreteTransferFcn: '<S1>/ValveDynamicsInverse' *)

        IF rtb_Switch3 <> 0.0 THEN 
            ValveDynamicsInverse_states[0] := 0.0;
            ValveDynamicsInverse_states[1] := 0.0;
        END_IF;

        rtb_Switch3 := (fPressureFeedback - (ValveDynamicsInverse_states[0] * VectorConcatenate3[1])) - (ValveDynamicsInverse_states[1] * VectorConcatenate3[2]);
        (* Switch: '<S1>/Switch2' incorporates:
         *  Constant: '<S1>/Constant'
         *  DiscreteTransferFcn: '<S1>/ValveDynamicsInverse' *)

        IF bEnable THEN 
            fPressureFeedback := ((VectorConcatenate2[0] * rtb_Switch3) + (ValveDynamicsInverse_states[0] * VectorConcatenate2[1])) + (ValveDynamicsInverse_states[1] * VectorConcatenate2[2]);
        ELSE 
            fPressureFeedback := 0.0;
        END_IF;

        (* End of Switch: '<S1>/Switch2' *)
        

        (* Saturate: '<S1>/Saturation5' *)

        IF fPressureFeedback > 1.0 THEN 
            (* Outport: '<Root>/fPressureFeedback' *)
            fPressureFeedback := 1.0;
        ELSIF fPressureFeedback < -1.0 THEN 
            (* Outport: '<Root>/fPressureFeedback' *)
            fPressureFeedback := -1.0;
        END_IF;

        (* End of Saturate: '<S1>/Saturation5' *)
        

        (* Update for DiscreteTransferFcn: '<S1>/HighPassFilter' *)
        HighPassFilter_states := HighPassFilter_tmp;
        (* Update for DiscreteTransferFcn: '<S1>/ValveDynamicsInverse' *)
        ValveDynamicsInverse_states[1] := ValveDynamicsInverse_states[0];
        ValveDynamicsInverse_states[0] := rtb_Switch3;
        (* End of Outputs for SubSystem: '<Root>/FB_ActiveDamping' *)
END_CASE;

END_FUNCTION_BLOCK

// ---- POUs/Programs/P_CraneControl.TcPOU
PROGRAM P_CraneControl
VAR
	fbTime				:	FB_Clock;
	fbSetMode			:	FB_SetMode;
	fbManualControl 	:	FB_ManualControl;
	fbAutomaticControl	:	FB_AutomaticControl;
	fbActiveDamping		:	FB_ActiveDamping;
	stActiveDamping		:	ST_ActiveDamping;
	fbCraneSimulator	:	FB_CraneSimulator;
	
	eMode 		:	E_Mode;
	fControlOutputNormalized : LREAL;
END_VAR

fbCraneSimulator
(
	ssMethodType := BOOL_TO_SINT(G_Parameter.bEnableSimulation),
	uDCV := G_Input.fJoyStickSignal,
);
	
	

fbTime
(
	bStart := G_Input.bStartSwitch,
	bStop := G_Input.bStopSwitch,
	fCycleTime := G_Parameter.fCycleTime,
	fTimeInSeconds => G_Parameter.fTime
	
);
	
fbSetMode
(
	bPower := G_Input.bPoweSwitch,
	bOn := G_Input.bOnOffSwitch,
	bMode := G_Input.bModeSwitch,
	bStart := G_Input.bStartSwitch,
	bStop := G_Input.bStopSwitch,
	eMode => G_Parameter.eMode,
	bGreenLight => G_Output.bGreenLed,
	bRedLight => G_Output.bRedLed,
	sMode => G_Output.sModeDisplay	
);


IF G_Input.bPoweSwitch = FALSE OR G_Input.bOnOffSwitch = FALSE OR G_Input.bStopSwitch = TRUE THEN
	G_Input.bStartSwitch := FALSE;
	G_Input.bStopSwitch := FALSE;
END_IF


fbManualControl(
	bEnable := (G_Parameter.eMode = E_Mode.Manual),
	eMode := eMode,
	fJoyStickInput := G_Input.fJoyStickSignal,
	fManualControlOutput => G_Output.fOpenLoopControlOutput
);


fbAutomaticControl(
	bEnable := (G_Parameter.eMode = E_Mode.Auto),
	eMode := eMode,
	bStartSwitch := G_Input.bStartSwitch,
	bStopSwitch := G_Input.bStopSwitch
	);
	
	
	
	
	
fbActiveDamping(
	ssMethodType := BOOL_TO_SINT(G_Parameter.bEnableActiveDamping),
	bEnable := G_Input.bStartSwitch,
	fPressurePistonSide_Pa := fbCraneSimulator.ppbar,
	fPressureRodSide_Pa := fbCraneSimulator.prbar,
	fkQfInv := stActiveDamping.fFlowGainInverse,
	HPF_Num1 := stActiveDamping.fHPF_Num1,
	HPF_Num2 := stActiveDamping.fHPF_Num2,
	HPF_Den1 := stActiveDamping.fHPF_Den1,
	HPF_Den2 := stActiveDamping.fHPF_Den2,
	VDI_Num1 := stActiveDamping.fVDI_Num1,
	VDI_Num2 := stActiveDamping.fVDI_Num2,
	VDI_Num3 := stActiveDamping.fVDI_Num3,
	VDI_Den1 := stActiveDamping.fVDI_Den1,
	VDI_Den2 := stActiveDamping.fVDI_Den2,
	VDI_Den3 := stActiveDamping.fVDI_Den3,
);



IF (G_parameter.eMode = E_Mode.Manual AND G_Input.bStartSwitch = TRUE) THEN
	fControlOutputNormalized := LIMIT(-1.0, (fbManualControl.fManualControlOutput - fbActiveDamping.fPressureFeedback), 1.0);
ELSIF (G_Parameter.eMode = E_Mode.Auto AND G_Input.bStartSwitch = TRUE) THEN
	fControlOutputNormalized := LIMIT(-1.0, (fbAutomaticControl.fAutoOutput - fbActiveDamping.fPressureFeedback), 1.0);
ELSE
	fControlOutputNormalized := 0.0;
END_IF

END_PROGRAM

// ---- GlobalTextList.TcGTLO
TEXTLIST GlobalTextList
  698 = '%f'
  490 = '%r'
  972 = '%s'
  141 = 'AUTO'
  747 = 'JOYSTICK'
  947 = 'MANUAL'
  454 = 'OFF'
  689 = 'ON'
  906 = 'OUTPUT SIGNAL TO CONTROL VALVE'
  879 = 'POWER'
  629 = 'Pressure feedback'
  764 = 'Simulator xm'
  724 = 'START'
  618 = 'STOP'
  880 = 'Velocity Feed Forward'
END_TEXTLIST

// ---- VISUs/HMI.TcVIS
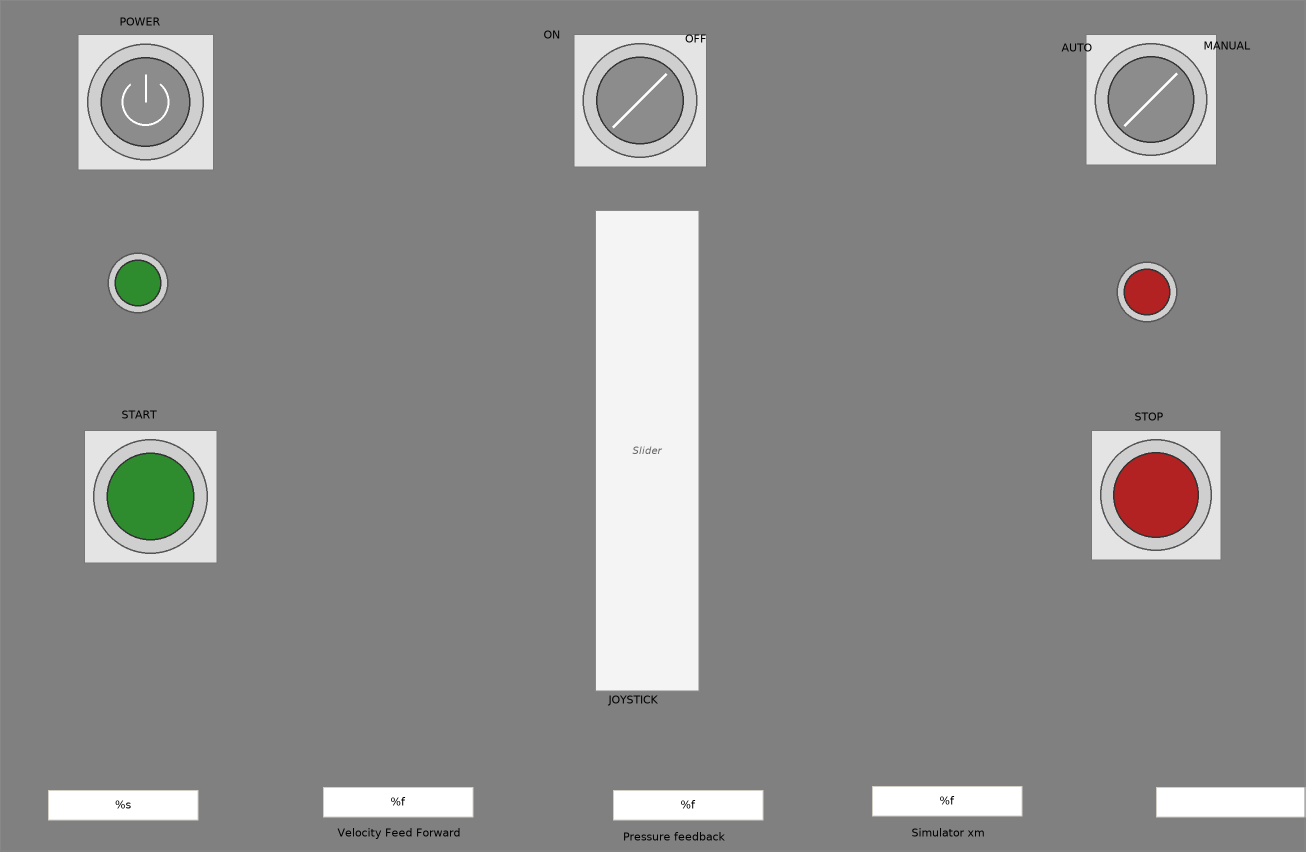
VISUALIZATION HMI  // 1306x852
    PowerSwitch (75,34 141x136), variable: G_Input.bPoweSwitch, behaviour: TOGGLE, style: Switch-PowerSwitch-Gray
    PushSwitch (74,430 153x133), variable: G_Input.bStartSwitch, behaviour: TOGGLE, style: Switch-PushSwitch-Green
    PushSwitch (1085,430 142x130), variable: G_Input.bStopSwitch, behaviour: TOGGLE, style: Switch-PushSwitch-Red
    RotarySwitch (566,34 148x133), variable: G_Input.bOnOffSwitch, behaviour: TOGGLE, style: Switch-RotarySwitch-Gray
    RotarySwitch (1085,34 132x131), variable: G_Input.bModeSwitch, behaviour: TOGGLE, style: Switch-RotarySwitch-Gray
    Slider (595,210 104x481), variable: G_Input.fJoyStickSignal, scale -1..1
    Label (1002,33 150x30), "AUTO"
    Label (1074,402 150x30), "STOP"
    Label (1152,31 150x30), "MANUAL"
    Label (477,20 150x30), "ON"
    Label (621,24 150x30), "OFF"
    Label (64,400 150x30), "START"
    Label (65,7 150x30), "POWER"
    Lamp1 (103,248 70x70), variable: G_Output.bGreenLed, style: Lamp-Lamp1-Green
    Lamp1 (1112,257 70x70), variable: G_Output.bRedLed, style: Lamp-Lamp1-Red
    Textfield (323,787 150x30), "%f", text variable: G_Output.fOpenLoopControlOutput
    Label (251,818 296x30), "Velocity Feed Forward"
    Label (558,685 150x30), "JOYSTICK"
    Textfield (48,790 150x30), "%s", text variable: G_Output.sModeDisplay
    Textfield (613,790 150x30), "%f", text variable: P_CraneControl.fbActiveDamping.fPressureFeedback
    Textfield (872,786 150x30), "%f", text variable: P_CraneControl.fbCraneSimulator.xm
    Textfield (1156,787 150x30)
    Label (599,822 150x30), "Pressure feedback"
    Label (873,818 150x30), "Simulator xm"
END_VISUALIZATION
